(* Logix 5000 project; controller ToyPlant Emulate 5570 rev 30.12; software revision 30.00 *)

TASK MainTask (continuous, watchdog 500 ms) : MainProgram

MODULES
   Local : Emulate 5570 (ICP 2, rev 30.12)
      VIRTUAL_INPUTS : vendor 1 type 0 code 15 (ICP 3, rev 1.1, Output RPI 50 ms)
END_MODULES

PROGRAM MainProgram   (* main routine MotoEnsamble *)
VAR
   Action_001 : SFC_ACTION := (Status := 16#c020_0000, A := 1, Q := 1, PauseTimer := 1, Count := 2);
   Action_009 : SFC_ACTION := (Status := 16#0020_0000, PauseTimer := 1, Count := 1);
   Action_010 : SFC_ACTION := (Status := 16#c020_0000, A := 1, Q := 1, PauseTimer := 1, Count := 2);
   Action_011 : SFC_ACTION := (Status := 16#0020_0000, PauseTimer := 1, Count := 1);
   Action_012 : SFC_ACTION := (Status := 16#0020_0000, PauseTimer := 1, Count := 1);
   Action_013 : SFC_ACTION := (Status := 16#0020_0000, PauseTimer := 1, Count := 1);
   Action_014 : SFC_ACTION := (Status := 16#0020_0000, PauseTimer := 1, Count := 1);
   Action_015 : SFC_ACTION := (Status := 16#0020_0000, PauseTimer := 1, Count := 1);
   Action_016 : SFC_ACTION := (Status := 16#0020_0000, PauseTimer := 1, Count := 1);
   Action_017 : SFC_ACTION := (Status := 16#0020_0000, PauseTimer := 1, Count := 1);
   StartEnsamble : ALIAS FOR Local:3:I.Data[1].0;
   Step_000 : SFC_STEP := (Status := 16#a820_0201, X := 1, SA := 1, DN := 1, PauseTimer := 1, T := 31632, TMax := 31632, Count := 2);
   Step_006 : SFC_STEP := (Status := 16#0020_0000, PauseTimer := 1);
   Step_007 : SFC_STEP := (Status := 16#a820_0201, X := 1, SA := 1, DN := 1, PauseTimer := 1, T := 31632, TMax := 31632, Count := 2);
   Step_008 : SFC_STEP := (Status := 16#0820_0001, DN := 1, PauseTimer := 1, T := 2120, TMax := 2120, Count := 1);
   Step_009 : SFC_STEP := (Status := 16#0820_0001, DN := 1, PauseTimer := 1, T := 6321, TMax := 6321, Count := 1);
   Step_010 : SFC_STEP := (Status := 16#0820_0001, DN := 1, PauseTimer := 1, T := 741, TMax := 741, Count := 1);
   Step_011 : SFC_STEP := (Status := 16#0820_0001, DN := 1, PauseTimer := 1, T := 933, TMax := 933, Count := 1);
   Step_012 : SFC_STEP := (Status := 16#0820_0001, DN := 1, PauseTimer := 1, T := 527, TMax := 527, Count := 1);
   TimerChasis : FBD_TIMER := (TimerEnable := 1, PRE := 700, ACC := 720, EN := 1, DN := 1);
   TimerPuertaAbierta : FBD_TIMER := (TimerEnable := 1, PRE := 900, ACC := 912, EN := 1, DN := 1);
   TimerPuertaCerrada : FBD_TIMER := (TimerEnable := 1, PRE := 500, ACC := 500, EN := 1, DN := 1);
   Tran_000 : BOOL;
   Tran_007 : BOOL;
   Tran_008 : BOOL := 1;
   Tran_009 : BOOL := 1;
   Tran_010 : BOOL := 1;
   Tran_011 : BOOL := 1;
   Tran_012 : BOOL := 1;
END_VAR
VAR_OUTPUT
   CerrarPuertaMoto : BOOL := 1; {access Read Only}
   Chasis_0 : BOOL := 1;
   Chasis_1 : BOOL := 1;
   RuedaDelantera_0 : BOOL := 1;
   RuedaDelantera_1 : BOOL := 1;
   RuedaDelantera_2 : BOOL := 1;
   RuedaTrasera_0 : BOOL := 1;
   RuedaTrasera_1 : BOOL := 1;
   RuedaTrasera_2 : BOOL := 1;
END_VAR
VAR_INPUT
   Sensor_RuedaDelantera1 : BOOL;
   Sensor_RuedaDelantera2 : BOOL;
   Sensor_RuedaTrasera1 : BOOL;
   Sensor_RuedaTrasera2 : BOOL;
   SensorChasis : BOOL;
END_VAR

ROUTINE MainRoutine   (* sequential function chart *)
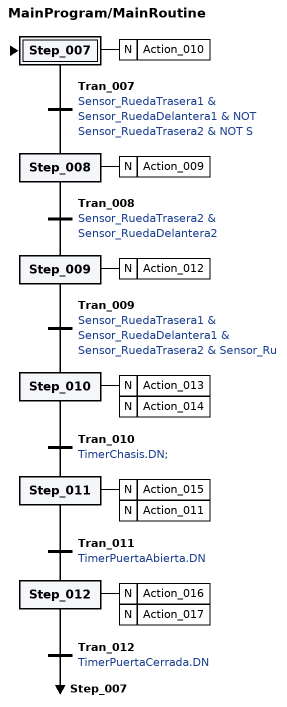
   INITIAL_STEP Step_007:
      ACTION Action_010 (N):
         CerrarPuertaMoto := 1;
      END_ACTION
   END_STEP
   TRANSITION Tran_007 FROM Step_007 TO Step_008
      := Sensor_RuedaTrasera1 & Sensor_RuedaDelantera1 & NOT Sensor_RuedaTrasera2 & NOT Sensor_RuedaDelantera2 & CerrarPuertaMoto
         
   END_TRANSITION
   STEP Step_008:
      ACTION Action_009 (N):
         RuedaDelantera_1 := 1;
         RuedaTrasera_1 := 1;
      END_ACTION
   END_STEP
   TRANSITION Tran_008 FROM Step_008 TO Step_009
      := Sensor_RuedaTrasera2 & Sensor_RuedaDelantera2
         
   END_TRANSITION
   STEP Step_009:
      ACTION Action_012 (N):
         RuedaTrasera_0 := 1;
         RuedaDelantera_0 := 1;
      END_ACTION
   END_STEP
   TRANSITION Tran_009 FROM Step_009 TO Step_010
      := Sensor_RuedaTrasera1 & Sensor_RuedaDelantera1 & Sensor_RuedaTrasera2 & Sensor_RuedaDelantera2 & SensorChasis
   END_TRANSITION
   STEP Step_010:
      ACTION Action_013 (N):
         Chasis_1 := 1;
      END_ACTION
      ACTION Action_014 (N):
         TimerChasis.TimerEnable := 1;
         TONR(TimerChasis);
         TimerChasis.PRE := 700;
         
      END_ACTION
   END_STEP
   TRANSITION Tran_010 FROM Step_010 TO Step_011
      := TimerChasis.DN;
   END_TRANSITION
   STEP Step_011:
      ACTION Action_015 (N):
         RuedaTrasera_2 := 1;
         RuedaDelantera_2 := 1;
      END_ACTION
      ACTION Action_011 (N):
         TimerPuertaAbierta.TimerEnable := 1;
         TONR(TimerPuertaAbierta);
         TimerPuertaAbierta.PRE := 900;
         
      END_ACTION
   END_STEP
   TRANSITION Tran_011 FROM Step_011 TO Step_012
      := TimerPuertaAbierta.DN
   END_TRANSITION
   STEP Step_012:
      ACTION Action_016 (N):
         CerrarPuertaMoto := 0;
         RuedaTrasera_0 := 1;
         RuedaDelantera_0 := 1;
         Chasis_0 :=1;
      END_ACTION
      ACTION Action_017 (N):
         TimerPuertaCerrada.TimerEnable := 1;
         TONR(TimerPuertaCerrada);
         TimerPuertaCerrada.PRE := 500;
         
      END_ACTION
   END_STEP
   TRANSITION Tran_012 FROM Step_012 TO Step_007
      := TimerPuertaCerrada.DN
   END_TRANSITION
END_ROUTINE

ROUTINE MotoEnsamble   (* sequential function chart *)
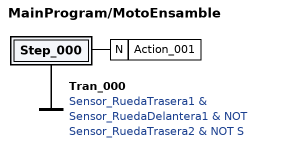
   INITIAL_STEP Step_000:
      ACTION Action_001 (N):
         CerrarPuertaMoto := 1;
      END_ACTION
   END_STEP
   TRANSITION Tran_000 FROM Step_000 TO ()
      := Sensor_RuedaTrasera1 & Sensor_RuedaDelantera1 & NOT Sensor_RuedaTrasera2 & NOT Sensor_RuedaDelantera2 & CerrarPuertaMoto
         
   END_TRANSITION
END_ROUTINE
END_PROGRAM
